(* CoDeSys 2.3 export: VISUPORTESET2.EXP *)

(* POU Simulation_Visuelle/VisuPortesET2, ST *)
FUNCTION VisuPortesET2 : BOOL
VAR_INPUT
END_VAR
VAR
	TimerDeTempo: TP;
	CompteurPortesVisu: INT;
	CompteurVarVisu: INT;
	CompteurDeTemps: INT;
	Step: INT;
	CompteurLocal: INT;
	CONTACTEUR_SEC: INT;
END_VAR
(* Cette fonction sert à fermer les portes de l'etage 2 en fonction des donné transmises par le porgramme principal*

	La fonction va simuler une fermeture sur action d'un moteur, et simuler le capteur  lorsque la coordonée de position fermé est atteinte : x=0 et y=-2*)
IF F2 OR O2 THEN
	(*On simule la position physique du contacteur avec des coordonnées*)
	IF F2 THEN CONTACTEUR_SEC:=-71;
	ELSE CONTACTEUR_SEC:=0;END_IF
	wait(IN:=TRUE, PT:=T#1ms);
	FOR CompteurLocal:=1 TO 3 BY 1 DO
		IF NOT wait.Q THEN
			wait(IN:=FALSE);
			(* en fonction de l'état du contacteur nous allons
			simuler une ouverture/fermeture de la porte*)

			(* nous allons utiliser les fonctions de coordonnées
			pour que la simulation suivent une trajectoire excate et soienet parfaitement synchronisé*)
			IF VisuET2Dx > CONTACTEUR_SEC THEN
				VisuET2Dx:=VisuET2Dx-1;
				VisuET2Dy:=FX_PorteD(VisuET2Dx);
				VisuET2Gx:=FX_Porte_Vitesse(VisuET2Dx);
				VisuET2Gy:=FX_PorteG(VisuET2Gx);
			ELSIF  VisuET2Dx < CONTACTEUR_SEC THEN
				VisuET2Dx:=VisuET2Dx+1;
				VisuET2Dy:=FX_PorteD(VisuET2Dx);
				VisuET2Gx:=FX_Porte_Vitesse(VisuET2Dx);
				VisuET2Gy:=FX_PorteG(VisuET2Gx);
			END_IF
		END_IF
	END_FOR
END_IF

IF VisuET2Dx = - 71  THEN P2fer:=TRUE;
ELSE P2fer:=FALSE;END_IF

IF VisuET2Dx = 0  THEN P2ouv:=TRUE;
ELSE P2ouv:=FALSE;END_IF
END_FUNCTION
